// Gets the lower bound index of the array of specified type.
FUNCTION F_GetULIntArrayLowerBound : T_Position // The lower bound index of the specified array.
VAR_IN_OUT
	arArray : ARRAY[*] OF ULINT; // The array to query.
END_VAR

F_GetULIntArrayLowerBound := LOWER_BOUND(arArray, 1);

END_FUNCTION

(* stored: Version 1.1.0.1
   POU F_GetULIntArrayLowerBound: Id {e6552f3e-d2ae-0a3d-3e13-d095b72ebf4a}, SpecialFunc None *)
